(* CODESYS project canbus.new.api.20190227.2_RECOVERED_2019-08-13T14-24-19.project
   Description: Receives some incoming messages and echoes them with CAN-ID +1
   Company: 3S - Smart Software Solutions GmbH
   Version: 1.0.0.0
   Title: CAN Bus API Example
   Author: 3S - Smart Software Solutions GmbH

Project tree, tasks and I/O mapping:
  Device : Changsha-Cyber-MI-linux, Changsha Cyber-MI Co., Ltd., version 3.5.10.40
    application Application
      libraries: CAN API, 1.0.0.3 (3S - Smart Software Solutions GmbH); Standard, * (System); CAA CiA 405, * (CAA Technical Workgroup)
      task MainTask (cyclic, interval t#20ms, priority 1) calls ST_PRG
      ST Example/
        function block MsgProcessor_EchoST [ST]: ProcessMessage
        program ST_PRG [ST]
      global variables GVL
      CFC Example/
        function block MsgProcessor_EchoCFC [CFC]: ProcessMessage
        program CFC_PRG [CFC]
    SoftMotion General Axis Pool
    CANbus_1 : CANbus, 3S - Smart Software Solutions GmbH, version 3.5.12.0
      CANopen_Manager : CANopen_Manager, 3S - Smart Software Solutions GmbH, version 3.5.10.0
          settings: ConfigVersion = 50659584
        Singleturn_Encoder_M36X8 : Singleturn Encoder M36X8, Kuebler GmbH, order no. 8.M36X8.XXCX.211X, version Revision=16#00000006, FileVersion=1.5
            settings: NODEIDSAVED = 1; SDO Timeout = 1000000; EXPERTSETTINGS = FALSE; Heartbeat-Producer Time = 200; PDO 16#1800.COBID = 16#00000181; Process by CANopenManager = TRUE; PDO 16#1801.COBID = 16#00000281; PDO 16#1801.Transmission Type = 16#01; Process by CANopenManager = TRUE; PDO 16#1802.COBID = 16#00000381; Process by CANopenManager = TRUE; Position Value.Subindex = 16#00; Speed Value 1.Subindex = 16#01; Position Value.Subindex = 16#00; SDO List.Set Guardtime.Index = 16#100C; SDO List.Set Guardtime.Subindex = 16#00; SDO List.Set Guardtime.Value = 16#00000000; SDO List.Set Guardtime.Size = 16; SDO List.Set Guardtime.AbortIfError = FALSE; SDO List.Set Guardtime.JumpToLine = FALSE; SDO List.Set Guardtime.Line = 0; SDO List.Set Lifetime.Index = 16#100D; SDO List.Set Lifetime.Subindex = 16#00; SDO List.Set Lifetime.Value = 16#00000000; SDO List.Set Lifetime.Size = 8; SDO List.Set Lifetime.AbortIfError = FALSE; SDO List.Set Lifetime.JumpToLine = FALSE; SDO List.Set Lifetime.Line = 0; SDO List.Set Heartbeat Producer.Index = 16#1017; SDO List.Set Heartbeat Producer.Subindex = 16#00; SDO List.Set Heartbeat Producer.Value = 16#000000C8; SDO List.Set Heartbeat Producer.Size = 16; SDO List.Set Heartbeat Producer.AbortIfError = FALSE; SDO List.Set Heartbeat Producer.JumpToLine = FALSE; SDO List.Set Heartbeat Producer.Line = 0; SDO List.Disable PDO.Index = 16#1800; SDO List.Disable PDO.Subindex = 16#01; SDO List.Disable PDO.Value = 16#80000181; SDO List.Disable PDO.Size = 32; SDO List.Disable PDO.AbortIfError = FALSE;
              SDO List.Disable PDO.JumpToLine = FALSE; SDO List.Disable PDO.Line = 0; SDO List.Set transmission type.Index = 16#1800; SDO List.Set transmission type.Subindex = 16#02; SDO List.Set transmission type.Value = 16#FF; SDO List.Set transmission type.Size = 8; SDO List.Set transmission type.AbortIfError = FALSE; SDO List.Set transmission type.JumpToLine = FALSE; SDO List.Set transmission type.Line = 0; SDO List.Set inhibit time.Index = 16#1800; SDO List.Set inhibit time.Subindex = 16#03; SDO List.Set inhibit time.Value = 16#0000; SDO List.Set inhibit time.Size = 16; SDO List.Set inhibit time.AbortIfError = FALSE; SDO List.Set inhibit time.JumpToLine = FALSE; SDO List.Set inhibit time.Line = 0; SDO List.Set event time.Index = 16#1800; SDO List.Set event time.Subindex = 16#05; SDO List.Set event time.Value = 16#0000; SDO List.Set event time.Size = 16; SDO List.Set event time.AbortIfError = FALSE; SDO List.Set event time.JumpToLine = FALSE; SDO List.Set event time.Line = 0; SDO List.Clear pdo mapping.Index = 16#1A00; SDO List.Clear pdo mapping.Subindex = 16#00; SDO List.Clear pdo mapping.Value = 16#0; SDO List.Clear pdo mapping.Size = 8; SDO List.Clear pdo mapping.AbortIfError = FALSE; SDO List.Clear pdo mapping.JumpToLine = FALSE; SDO List.Clear pdo mapping.Line = 0; SDO List.Set Mapping.Index = 16#1A00; SDO List.Set Mapping.Subindex = 16#01; SDO List.Set Mapping.Value = 16#60040020; SDO List.Set Mapping.Size = 32; SDO List.Set Mapping.AbortIfError = FALSE; SDO List.Set Mapping.JumpToLine = FALSE; SDO List.Set Mapping.Line = 0; SDO List.Set number of mappings.Index = 16#1A00; SDO List.Set number of mappings.Subindex = 16#00; SDO List.Set number of mappings.Value = 16#01;
              SDO List.Set number of mappings.Size = 8; SDO List.Set number of mappings.AbortIfError = FALSE; SDO List.Set number of mappings.JumpToLine = FALSE; SDO List.Set number of mappings.Line = 0; SDO List.Set and enable COB-ID.Index = 16#1800; SDO List.Set and enable COB-ID.Subindex = 16#01; SDO List.Set and enable COB-ID.Value = 16#00000181; SDO List.Set and enable COB-ID.Size = 32; SDO List.Set and enable COB-ID.AbortIfError = FALSE; SDO List.Set and enable COB-ID.JumpToLine = FALSE; SDO List.Set and enable COB-ID.Line = 0; SDO List.Disable PDO.Index = 16#1801; SDO List.Disable PDO.Subindex = 16#01; SDO List.Disable PDO.Value = 16#80000281; SDO List.Disable PDO.Size = 32; SDO List.Disable PDO.AbortIfError = FALSE; SDO List.Disable PDO.JumpToLine = FALSE; SDO List.Disable PDO.Line = 0; SDO List.Set transmission type.Index = 16#1801; SDO List.Set transmission type.Subindex = 16#02; SDO List.Set transmission type.Value = 16#01; SDO List.Set transmission type.Size = 8; SDO List.Set transmission type.AbortIfError = FALSE; SDO List.Set transmission type.JumpToLine = FALSE; SDO List.Set transmission type.Line = 0; SDO List.Set inhibit time.Index = 16#1801; SDO List.Set inhibit time.Subindex = 16#03; SDO List.Set inhibit time.Value = 16#0000; SDO List.Set inhibit time.Size = 16; SDO List.Set inhibit time.AbortIfError = FALSE; SDO List.Set inhibit time.JumpToLine = FALSE; SDO List.Set inhibit time.Line = 0; SDO List.Set event time.Index = 16#1801; SDO List.Set event time.Subindex = 16#05; SDO List.Set event time.Value = 16#0000; SDO List.Set event time.Size = 16; SDO List.Set event time.AbortIfError = FALSE; SDO List.Set event time.JumpToLine = FALSE; SDO List.Set event time.Line = 0; SDO List.Clear pdo mapping.Index = 16#1A01;
              SDO List.Clear pdo mapping.Subindex = 16#00; SDO List.Clear pdo mapping.Value = 16#0; SDO List.Clear pdo mapping.Size = 8; SDO List.Clear pdo mapping.AbortIfError = FALSE; SDO List.Clear pdo mapping.JumpToLine = FALSE; SDO List.Clear pdo mapping.Line = 0; SDO List.Set Mapping.Index = 16#1A01; SDO List.Set Mapping.Subindex = 16#01; SDO List.Set Mapping.Value = 16#60300110; SDO List.Set Mapping.Size = 32; SDO List.Set Mapping.AbortIfError = FALSE; SDO List.Set Mapping.JumpToLine = FALSE; SDO List.Set Mapping.Line = 0; SDO List.Set number of mappings.Index = 16#1A01; SDO List.Set number of mappings.Subindex = 16#00; SDO List.Set number of mappings.Value = 16#01; SDO List.Set number of mappings.Size = 8; SDO List.Set number of mappings.AbortIfError = FALSE; SDO List.Set number of mappings.JumpToLine = FALSE; SDO List.Set number of mappings.Line = 0; SDO List.Set and enable COB-ID.Index = 16#1801; SDO List.Set and enable COB-ID.Subindex = 16#01; SDO List.Set and enable COB-ID.Value = 16#00000281; SDO List.Set and enable COB-ID.Size = 32; SDO List.Set and enable COB-ID.AbortIfError = FALSE; SDO List.Set and enable COB-ID.JumpToLine = FALSE; SDO List.Set and enable COB-ID.Line = 0; SDO List.Disable PDO.Index = 16#1802; SDO List.Disable PDO.Subindex = 16#01; SDO List.Disable PDO.Value = 16#80000381; SDO List.Disable PDO.Size = 32; SDO List.Disable PDO.AbortIfError = FALSE; SDO List.Disable PDO.JumpToLine = FALSE; SDO List.Disable PDO.Line = 0; SDO List.Set transmission type.Index = 16#1802; SDO List.Set transmission type.Subindex = 16#02; SDO List.Set transmission type.Value = 16#FF; SDO List.Set transmission type.Size = 8; SDO List.Set transmission type.AbortIfError = FALSE; SDO List.Set transmission type.JumpToLine = FALSE;
              SDO List.Set transmission type.Line = 0; SDO List.Set inhibit time.Index = 16#1802; SDO List.Set inhibit time.Subindex = 16#03; SDO List.Set inhibit time.Value = 16#0000; SDO List.Set inhibit time.Size = 16; SDO List.Set inhibit time.AbortIfError = FALSE; SDO List.Set inhibit time.JumpToLine = FALSE; SDO List.Set inhibit time.Line = 0; SDO List.Set event time.Index = 16#1802; SDO List.Set event time.Subindex = 16#05; SDO List.Set event time.Value = 16#0000; SDO List.Set event time.Size = 16; SDO List.Set event time.AbortIfError = FALSE; SDO List.Set event time.JumpToLine = FALSE; SDO List.Set event time.Line = 0; SDO List.Clear pdo mapping.Index = 16#1A02; SDO List.Clear pdo mapping.Subindex = 16#00; SDO List.Clear pdo mapping.Value = 16#0; SDO List.Clear pdo mapping.Size = 8; SDO List.Clear pdo mapping.AbortIfError = FALSE; SDO List.Clear pdo mapping.JumpToLine = FALSE; SDO List.Clear pdo mapping.Line = 0; SDO List.Set Mapping.Index = 16#1A02; SDO List.Set Mapping.Subindex = 16#01; SDO List.Set Mapping.Value = 16#60040020; SDO List.Set Mapping.Size = 32; SDO List.Set Mapping.AbortIfError = FALSE; SDO List.Set Mapping.JumpToLine = FALSE; SDO List.Set Mapping.Line = 0; SDO List.Set number of mappings.Index = 16#1A02; SDO List.Set number of mappings.Subindex = 16#00; SDO List.Set number of mappings.Value = 16#01; SDO List.Set number of mappings.Size = 8; SDO List.Set number of mappings.AbortIfError = FALSE; SDO List.Set number of mappings.JumpToLine = FALSE; SDO List.Set number of mappings.Line = 0; SDO List.Set and enable COB-ID.Index = 16#1802; SDO List.Set and enable COB-ID.Subindex = 16#01; SDO List.Set and enable COB-ID.Value = 16#00000381; SDO List.Set and enable COB-ID.Size = 32;
              SDO List.Set and enable COB-ID.AbortIfError = FALSE; SDO List.Set and enable COB-ID.JumpToLine = FALSE; SDO List.Set and enable COB-ID.Line = 0; ConfigVersion = 50659584
            unmapped channels: Position Value, Speed Value 1, Position Value
*)

// Device/Application/GVL
VAR_GLOBAL
	(* Message count *)
	g_countMsg_resv_ST	: UINT;
	g_countMsg_send_ST	: UINT;
	
	g_countMsg_CFC	: UINT;
	
	(* This data type descripes the configuration of the CANbus Driver *)
	g_busConfig0		: CAN.DRIVER_CONFIG := (usiNetwork:= 0, uiBaudrate:= 250, ctMessages:= 100);
	
	g_busConfig1		: CAN.DRIVER_CONFIG := (usiNetwork:= 1, uiBaudrate:= 250, ctMessages:= 100);
 
	(* Time limit for receiving messages. T#0s:= no time limit *)
	g_tTimeLimit		: TIME := T#5MS;
	
END_VAR

// Device/Application/ST Example/ST_PRG
/// Receive all incoming messages and echos them with CobId +1
PROGRAM ST_PRG
VAR	
	(* A CANbus for handling 29bit CobIds *)
	driver0		: CAN.CANBus_29bit := (DriverConfig:= g_busConfig0);
	

	(* Handle for an Mask Receiver *)
	hMaskReceiver0	: CAN.CAA.HANDLE := CAN.CAA.gc_hINVALID;
		
	(* Received messages are passed to MessageProcessors. *)
	msgProcessor0	: MsgProcessor_EchoST;

	(* Defines a mask for the receiver *)
	maskConfig0		: CAN.RECEIVER_MASK := (
										dwIdValue:= 0, 
										dwIdMask:= 0, 
										xRTRValue:= FALSE, 
										xRTRMask:= FALSE, 
										x29BitIdValue:= TRUE, 
										x29BitIdMask:= FALSE, 
										xTransmitValue:= FALSE, 
										xTransmitMask:= TRUE, 
										xAlwaysNewest:= FALSE);
										
	message0 :CAN.MESSAGE;										

END_VAR

(***************************************************************)
//can 0

/// Configure the CAN Driver
driver0(DriverConfig:= g_busConfig0, eError=> );

/// Configure MessageProcessor
msgProcessor0(CANdriver:= driver0);

message0.udiCanID := 16#3A;
message0.usiDataLength := 8;
message0.xIs29BitMessage := TRUE;
message0.abyData[0] := 12;
message0.abyData[7] := 34;

driver0.SendMessage(message0, eError=>);
gvl.g_countMsg_send_ST := gvl.g_countMsg_send_ST + 1;

/// Create a Mask Receiver to receive all messages
/// Each call of GetMaskReceiver generates a new Receiver
IF hMaskReceiver0 = CAN.CAA.gc_hINVALID THEN
	hMaskReceiver0 := driver0.GetMaskReceiver(Mask:= maskConfig0, eError=> );
END_IF

/// Receive messages and hand them over to the MsgProccessor_Echo
driver0.ReceiveMessage(hReceiver:= hMaskReceiver0, itfMsgProcessor:= msgProcessor0, tTimeLimit:= g_tTimeLimit, eError=> );

END_PROGRAM

// Device/Application/ST Example/MsgProcessor_EchoST
/// MsgProcessor_Echo is the implimentation of IMessageProcessor. 
/// MsgProcessor_Echo simply counts all incoming messages and echos them with CobId +1
FUNCTION_BLOCK MsgProcessor_EchoST IMPLEMENTS CAN.IMessageProcessor
VAR_IN_OUT
	CANdriver	: CAN.CANBus_29bit;
END_VAR
VAR_OUTPUT
END_VAR
VAR
	_pCANdriver : POINTER TO CAN.CANBus_29bit;
END_VAR

_pCANdriver := ADR(CANdriver);

METHOD ProcessMessage
VAR_IN_OUT
	(* The messages received by the receiver *)
	Message	: CAN.RxMessage;
END_VAR
VAR
END_VAR
/// Echo incoming messages with CobId +1
IF _pCANdriver <> 0 THEN
	Message.udiCanId:= Message.udiCanID + 1;
//	_pCANdriver^.SendMessage(Message:= Message, eError=> );
	gvl.g_countMsg_resv_ST:= gvl.g_countMsg_resv_ST +1;
END_IF
END_METHOD

END_FUNCTION_BLOCK

// Device/Application/CFC Example/MsgProcessor_EchoCFC
FUNCTION_BLOCK MsgProcessor_EchoCFC IMPLEMENTS CAN.IMessageProcessor
VAR_IN_OUT
	CANdriver	: CAN.CANDriver_11bit;
END_VAR
VAR_OUTPUT
END_VAR
VAR
END_VAR

{attribute '''DOCU__COMMENT' := ' The Process Message Methode must be implementet by the user.'}
(* The Process Message Methode must be implementet by the user.*)
METHOD ProcessMessage
VAR_IN_OUT
	(* Incoming message *)
	Message	: CAN.RxMESSAGE;
END_VAR
VAR
	sender	: CAN.CANSender;
	xStart	: BOOL := TRUE;
	fTrig	: F_TRIG;
END_VAR
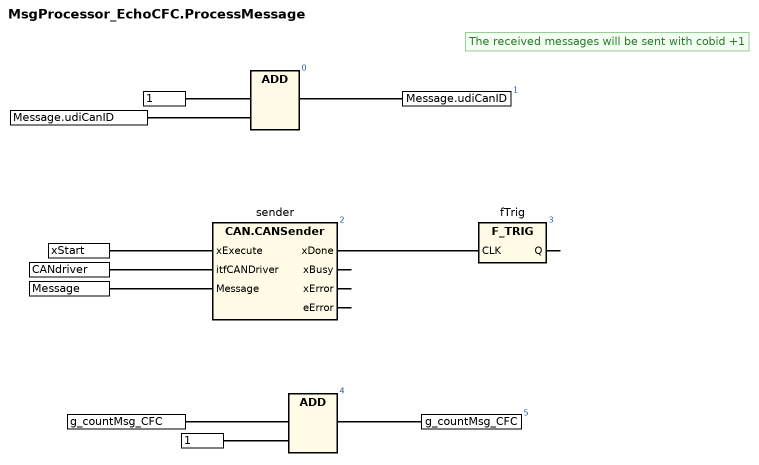
// The received messages will be sent with cobid +1
Message.udiCanID := 1 + Message.udiCanID;
sender(xExecute := xStart, itfCANDriver := CANdriver, Message := Message); // CAN.CANSender
fTrig(CLK := sender.xDone); // F_TRIG
g_countMsg_CFC := g_countMsg_CFC + 1;
END_METHOD

END_FUNCTION_BLOCK

// Device/Application/CFC Example/CFC_PRG
/// Receives messages with CobIds ranging from 16#500 to 16#550 and echoes them back with CobId +1
PROGRAM CFC_PRG
VAR
	driver11bit 	: CAN.CANDriver_11bit;
	                                
	areaReceiver	: CAN.CANAreaReceiver;
	singleReceiver	: CAN.CANSingleIdReceiver;
	diagnosis		: CAN.CANBusDiagnosis;
	
	msgProcessor	: MsgProcessor_EchoCFC;
END_VAR
VAR // added by the converter: edge detectors and wires of the graphical bodies
    _s1 : CAN.DRIVER_CONFIG;
    _s2 : CAN.RECEIVER_AREA;
    _s3 : CAN.RECEIVER_SINGLE_ID;
    _s4 : CAN.DIAGNOSIS_INFO;
END_VAR

// compose _s1 : CAN.DRIVER_CONFIG
_s1.usiNetwork := 0;
_s1.uiBaudrate := 500;
_s1.ctMessages := 100;
driver11bit(xEnable := TRUE, DriverConfig := _s1); // CAN.CANDriver_11bit
// compose _s2 : CAN.RECEIVER_AREA
_s2.dwIdStart := 16#500;
_s2.dwIdEnd := 16#550;
_s2.xRTRValue := false;
_s2.xRTRMask := false;
_s2.xTransmitValue := false;
_s2.xTransmitMask := true;
msgProcessor(CANdriver := driver11bit); // MsgProcessor_EchoCFC
areaReceiver(
    xEnable := driver11bit.xBusy,
    itfCANDriver := driver11bit,
    Area := _s2,
    itfMsgProcessor := msgProcessor,
    tTimeLimit := g_tTimeLimit); // CAN.CANAreaReceiver
diagnosis(xEnable := driver11bit.xBusy, itfCANDriver := driver11bit, DiagnosticInfo := _s4); // CAN.CANBusDiagnosis
// compose _s3 : CAN.RECEIVER_SINGLE_ID
_s3.dwCanId := 16#280;
_s3.xRTRValue := false;
_s3.xRTRMask := false;
_s3.x29BitIdValue := false;
_s3.x29BitIdMask := false;
_s3.xTransmitValue := false;
_s3.xTransmitMask := true;
_s3.xAlwaysNewest := false;
singleReceiver(
    xEnable := driver11bit.xBusy,
    itfCANDriver := driver11bit,
    itfMsgProcessor := msgProcessor,
    tTimeLimit := g_tTimeLimit,
    SingleId := _s3); // CAN.CANSingleIdReceiver
// compose _s4 : CAN.DIAGNOSIS_INFO

END_PROGRAM
